(* IEC 61131-3 sources: CodesysTest/export/SX_1195.dev/Plc Logic/Application/PRJ Specific/1195 Testing/DualMotorPressureBar_Async/FB_DualMotorPressureBar_Async.pou/IsIdle.prop, 1 file *)

(* ---- Get.pm.st ---- *)
(*#-#-#-#-#-#-#-#-#-#---Declaration---#-#-#-#-#-#-#-#-#-#-#-#-#*)

VAR
END_VAR
(*#-#-#-#-#-#-#-#-#-#---Implementation---#-#-#-#-#-#-#-#-#-#-#-#-#*)

IsIdle := (state = eDualMotorPressureBar_AsyncStates.Idle);
